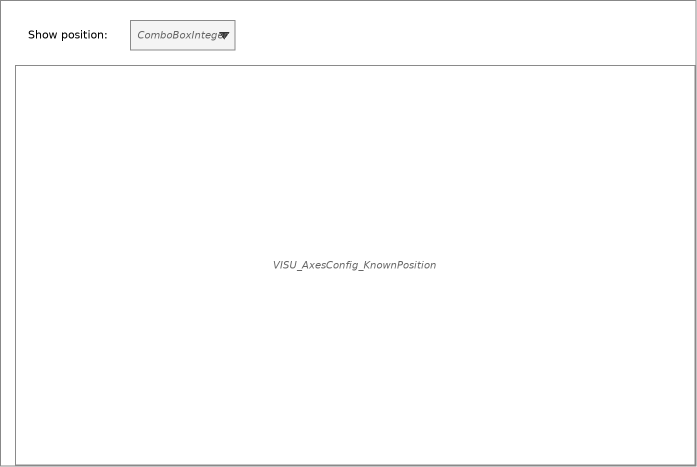
VISUALIZATION VISU_AxesConfig_KnownPositions  // 697x467
VAR_IN_OUT
    activePosition : INT;
    editable : AxesKnownPositionsConfig;
	active : AxesKnownPositionsConfig;
END_VAR
    Frame (15,65 680x400), frame switch variable: activePosition
        shows VISU_AxesConfig_KnownPosition(editable := editable.position0, active := active.position0)
        shows VISU_AxesConfig_KnownPosition(editable := editable.position1, active := active.position1)
        shows VISU_AxesConfig_KnownPosition(editable := editable.position2, active := active.position2)
        shows VISU_AxesConfig_KnownPosition(editable := editable.position3, active := active.position3)
        shows VISU_AxesConfig_KnownPosition(editable := editable.position4, active := active.position4)
        shows VISU_AxesConfig_KnownPosition(editable := editable.position5, active := active.position5)
        shows VISU_AxesConfig_KnownPosition(editable := editable.position6, active := active.position6)
        shows VISU_AxesConfig_KnownPosition(editable := editable.position7, active := active.position7)
        shows VISU_AxesConfig_KnownPosition(editable := editable.position8, active := active.position8)
        shows VISU_AxesConfig_KnownPosition(editable := editable.position9, active := active.position9)
        shows VISU_AxesConfig_KnownPosition(editable := editable.position10, active := active.position10)
        shows VISU_AxesConfig_KnownPosition(editable := editable.position11, active := active.position11)
        shows VISU_AxesConfig_KnownPosition(editable := editable.position12, active := active.position12)
        shows VISU_AxesConfig_KnownPosition(editable := editable.position13, active := active.position13)
        shows VISU_AxesConfig_KnownPosition(editable := editable.position14, active := active.position14)
        shows VISU_AxesConfig_KnownPosition(editable := editable.position15, active := active.position15)
        shows VISU_AxesConfig_KnownPosition(editable := editable.position16, active := active.position16)
        shows VISU_AxesConfig_KnownPosition(editable := editable.position17, active := active.position17)
        shows VISU_AxesConfig_KnownPosition(editable := editable.position18, active := active.position18)
        shows VISU_AxesConfig_KnownPosition(editable := editable.position19, active := active.position19)
    Label (25,20 150x30), "Show position:"
    ComboBoxInteger (130,20 105x30), variable: activePosition
END_VISUALIZATION

(* stored: Version 1.1.0.1, ProductVersion 3.1.4019.2
   Visu VISU_AxesConfig_KnownPositions: Id {9e6b4417-0d15-4fa9-b98a-627796a20d3d} *)
